PROGRAM POU
VAR
END_VAR

END_PROGRAM

(* stored: Version 1.1.0.1, ProductVersion 3.1.4024.13
   POU POU: Id {546a7c6c-c496-4c85-acb4-6897e0661962}, SpecialFunc None *)
